{attribute 'linkalways'} 
{attribute 'no_explicit_call' := 'This FB is a CLASS and must be accessed using methods or properties'}
{attribute 'enable_dynamic_creation'}
FUNCTION_BLOCK _ETcVnPixelPackMode EXTENDS EnumDatatypeBase
VAR
	localData : ETcVnPixelPackMode;
	activeData : REFERENCE TO ETcVnPixelPackMode;
	enumBaseDatatype : _BYTE(localData);
END_VAR

METHOD PRIVATE AddLocalEnumeration
VAR_INPUT
	Enumeration : T_MAXSTRING;
	Value : ETcVnPixelPackMode;
END_VAR
AddEnumeration(Enumeration, Value);
END_METHOD

PROPERTY PUBLIC Address : PVOID
GET
Address := ADR(activeData);
END_GET
END_PROPERTY

METHOD PUBLIC ClearReference
VAR_INPUT
END_VAR
activeData REF= localData;
SetBaseDatatypeReference();
END_METHOD

METHOD PUBLIC Clone : I_Datatype
VAR
    pClone : POINTER TO _ETcVnPixelPackMode;
END_VAR
pClone := __NEW(_ETcVnPixelPackMode(InitialValue := Value));
Clone := pClone^;
END_METHOD

METHOD FB_init : BOOL
VAR_INPUT
	bInitRetains : BOOL; // if TRUE, the retain variables are initialized (warm start / cold start)
	bInCopyCode : BOOL;  // if TRUE, the instance afterwards gets moved into the copy code (online change)
	InitialValue : ETcVnPixelPackMode;
END_VAR
localData := InitialValue;
AddBaseDatatype(enumBaseDatatype);
ClearReference();

AddLocalEnumeration('TCVN_PPM_NONE', ETcVnPixelPackMode.TCVN_PPM_NONE);
AddLocalEnumeration('TCVN_PPM_MONO1P', ETcVnPixelPackMode.TCVN_PPM_MONO1P);
AddLocalEnumeration('TCVN_PPM_MONO2P', ETcVnPixelPackMode.TCVN_PPM_MONO2P);
AddLocalEnumeration('TCVN_PPM_MONO4P', ETcVnPixelPackMode.TCVN_PPM_MONO4P);
AddLocalEnumeration('TCVN_PPM_MONO10PACKED', ETcVnPixelPackMode.TCVN_PPM_MONO10PACKED);
AddLocalEnumeration('TCVN_PPM_MONO12PACKED', ETcVnPixelPackMode.TCVN_PPM_MONO12PACKED);
AddLocalEnumeration('TCVN_PPM_RGB10V1PACKED', ETcVnPixelPackMode.TCVN_PPM_RGB10V1PACKED);
AddLocalEnumeration('TCVN_PPM_RGB10P32', ETcVnPixelPackMode.TCVN_PPM_RGB10P32);
AddLocalEnumeration('TCVN_PPM_RGB12V1PACKED', ETcVnPixelPackMode.TCVN_PPM_RGB12V1PACKED);
AddLocalEnumeration('TCVN_PPM_RGB565P', ETcVnPixelPackMode.TCVN_PPM_RGB565P);
AddLocalEnumeration('TCVN_PPM_BGR565P', ETcVnPixelPackMode.TCVN_PPM_BGR565P);
AddLocalEnumeration('TCVN_PPM_MONO10P', ETcVnPixelPackMode.TCVN_PPM_MONO10P);
AddLocalEnumeration('TCVN_PPM_MONO12P', ETcVnPixelPackMode.TCVN_PPM_MONO12P);
// AddLocalEnumeration('TCVN_PPM_MONO14P', ETcVnPixelPackMode.TCVN_PPM_MONO14P);
END_METHOD

PROPERTY PUBLIC Identifier : T_MAXSTRING
GET
Identifier := 'ETcVnPixelPackMode';
END_GET
END_PROPERTY

METHOD IsEnumeratorValueEqual : BOOL
VAR_INPUT
	Enumerator : I_KeyValueForwardEnumerator;
END_VAR
VAR
	storedValue : ETcVnPixelPackMode;
END_VAR
IF NOT Enumerator.TryGet(storedValue) THEN
	RETURN;
END_IF

IsEnumeratorValueEqual := storedValue = activeData;
END_METHOD

METHOD PUBLIC MakeReferenceTo
VAR_INPUT
	ReferenceTarget : REFERENCE TO ETcVnPixelPackMode;
END_VAR
activeData REF= ReferenceTarget;
SetBaseDatatypeReference();
END_METHOD

METHOD PROTECTED SetBaseDatatypeReference
VAR_INPUT
END_VAR
enumBaseDatatype.MakeReferenceTo(activeData);
END_METHOD

PROPERTY PUBLIC Size : UDINT
GET
Size := SIZEOF(activeData);
END_GET
END_PROPERTY

METHOD TryMakeReferenceTo : BOOL
VAR_INPUT
	Target : I_Datatype;
END_VAR
VAR
	pTargetData : POINTER TO ETcVnPixelPackMode;
END_VAR
IF NOT IsEquivalentTo(Target) THEN
	RETURN;
END_IF

pTargetData := Target.Address;
activeData REF= pTargetData^;
SetBaseDatatypeReference();
TryMakeReferenceTo := TRUE;
END_METHOD

PROPERTY PUBLIC Value : ETcVnPixelPackMode
GET
Value := activeData;
END_GET
SET
activeData := Value;
END_SET
END_PROPERTY

END_FUNCTION_BLOCK

(* stored: Version 1.1.0.1, ProductVersion 3.1.4026.19
   POU _ETcVnPixelPackMode: Id {d993a433-f6a2-41d8-9e7b-d4c38c49b5db}, SpecialFunc None
   Folder Core: Id {1b36a2da-cfcb-047d-0e3e-0d69b654cdf8}
   Folder Protected: Id {e1db430b-d611-0348-1253-28d827a38987}
   Folder Customize: Id {9ff60d3a-a1d2-050d-2ee1-84bc26a2ceff}
   Folder Constructor: Id {7b682f34-d669-4140-bb67-c6ff01de5e56}
   Folder Private: Id {6addf33c-582e-4555-b87b-f3eb8e51fc21}
   Folder Protected: Id {f2040aaf-28c8-40da-83ac-de62342aea23}
   Method AddLocalEnumeration: Id {20e09289-cd5b-4d32-b698-c4dc2e1e1079}
   Property Address: Id {d41e394a-90d1-05c5-1f38-1418b41956bd}
   Get Get: Id {6fcde248-3446-02ab-2511-029b56e3f0ab}
   Method ClearReference: Id {dcb3f578-1bfd-0447-16b1-7fa271cdefa6}
   Method Clone: Id {4f57a0f2-2730-4ffd-879a-3fb75b664491}
   Method FB_init: Id {e3b69484-84bb-47d6-8959-6fb3c14caba4}
   Property Identifier: Id {a68ec017-631f-4d64-a70a-61caa7666f18}
   Get Get: Id {c1c6cc72-b54e-4059-9e42-916fddf1e598}
   Method IsEnumeratorValueEqual: Id {a477fdc4-8b1e-4267-bc01-b44814d306fa}
   Method MakeReferenceTo: Id {064f95b9-4036-477e-a1fa-35659ca9107d}
   Method SetBaseDatatypeReference: Id {b23b6902-e441-068f-2b2d-477291a0b2d4}
   Property Size: Id {4186a091-c6b8-0dea-150d-93094c209f84}
   Get Get: Id {8621b9a4-80e4-03ef-33ee-afcb4b429fad}
   Method TryMakeReferenceTo: Id {08b15d71-a9b3-41f5-a1c3-124f0b463897}
   Property Value: Id {e8ec1d8b-5777-478d-bcc6-936369d97c71}
   Get Get: Id {89208553-e249-4602-bee2-300f45fd10e2}
   Set Set: Id {3743eb1f-2f45-47df-a180-99b520edaf62} *)
